Staubli VAL3: insertInstr.pgx

program insertInstr()
  local num i
  local string l_sMessage
  local num l_nIndex
  local string l_sItem
  local string l_sPath
begin
end
